// TIA Portal V17 export
// export: Created 2025-03-05T07:58:52.0345726Z, ExportSetting WithDefaults, DisplayName Totally Integrated Automation Portal, DisplayVersion V17 Update 8, DisplayName TIA Portal Openness, DisplayVersion V17 Update 8, DisplayName TIA Portal Version Control Interface, DisplayVersion V17, DisplayName SINAMICS Startdrive Advanced, DisplayVersion V17 SP2, DisplayName SINAMICS Startdrive G110M, G120, G120C, G120D, G120P, G115D, DisplayVersion V17 SP2, DisplayName SINAMICS Startdrive G130, G150, S120, S150, SINAMICS MV, S210, DisplayVersion V17 SP2, DisplayName STEP 7 Professional, DisplayVersion V17 Update 8, DisplayName SINUMERIK ONE STEP 7 Toolbox, DisplayVersion V17 Update 12, DisplayName SINUMERIK 840D sl STEP 7 Toolbox, DisplayVersion V17 Update 12, DisplayName STEP 7 Safety, DisplayVersion V17 Update 6, DisplayName WinCC Advanced, DisplayVersion V17 Update 8
DATA_BLOCK "LBP_HMI"   // DB19
TITLE = Operator panel signals / Señales panel de mando / Bedienfeld-Signale
{ S7_Optimized_Access := 'FALSE'; DB_Accessible_From_OPC_UA := 'FALSE' }
AUTHOR : SINUMERIK
FAMILY : SINUMERIK_ONE
VERSION : 6.15
// Interface between user program and operator panel, contains signals from/to the operating software. / Interfaz entre programa de usuario y panel de mando, contiene señales desde/hacia software operativo. / Schnittstelle zwischen Anwenderprogramm und Bedienfeld, enthält Signale von der/zu der Betriebssoftware.
// stored: AutoNumber false, DBAccessibleFromOPCUA false, DBAccessibleFromWebserver true, InstanceOfName LBP_typeHMI, InstanceOfType UDT, IsOnlyStoredInLoadMemory false, IsWriteProtectedInAS false
"LBP_typeHMI"
   // VAR RETAIN
   //    A_SCLight : Bool;
   //    A_SCDark : Bool;
   //    A_KeyDisable : Bool;
   //    A_ClearCanAl : Bool;
   //    A_ClearRecAl : Bool;
   //    f0_5 : Bool;
   //    A_SafeActionLog : Bool;
   //    A_ActWCS : Bool;
   //    A_PLCExtViewerReject : Bool;
   //    A_PLCExtViewerMode : Bool;
   //    f1_2 : Bool;
   //    f1_3 : Bool;
   //    f1_4 : Bool;
   //    f1_5 : Bool;
   //    f1_6 : Bool;
   //    f1_7 : Bool;
   //    A_1stError1 : Word;
   //    A_1stError2 : Word;
   //    A_ASpi1percent : Byte;
   //    A_ASpi2percent : Byte;
   //    A_MCPChan : Byte;
   //    A_OEM1 : Bool;
   //    A_OEM2 : Bool;
   //    A_AToolMeas : Bool;
   //    f9_3 : Bool;
   //    f9_4 : Bool;
   //    f9_5 : Bool;
   //    f9_6 : Bool;
   //    f9_7 : Bool;
   //    A_Hardkey : Byte;
   //    f11 : Byte;
   //    f12_0 : Bool;
   //    f12_1 : Bool;
   //    A_COM2 : Bool;
   //    A_COM1 : Bool;
   //    A_V24stop : Bool;
   //    A_V24ext : Bool;
   //    A_V24off : Bool;
   //    A_V24on : Bool;
   //    A_TeachDisable : Bool;
   //    f13_1 : Bool;
   //    f13_2 : Bool;
   //    f13_3 : Bool;
   //    f13_4 : Bool;
   //    A_PPdeload : Bool;
   //    A_PPload : Bool;
   //    A_PPsel : Bool;
   //    A_V24Index1 : Byte;
   //    A_V24Index2 : Byte;
   //    A_V24NoFile1 : Byte;
   //    A_V24NoFile2 : Byte;
   //    A_res18 : Byte;
   //    A_res19 : Byte;
   //    f20_0 : Bool;
   //    E_SCDark : Bool;
   //    E_Cancel : Bool;
   //    E_CanCleared : Bool;
   //    E_RecCleared : Bool;
   //    f20_5 : Bool;
   //    E_SimActiv : Bool;
   //    E_ActWCS : Bool;
   //    E_ActivWA : Byte;
   //    E_Chan : Byte;
   //    E_KeybHandl : Bool;
   //    E_DataTransf : Bool;
   //    E_DisplChange : Bool;
   //    f23_3 : Bool;
   //    f23_4 : Bool;
   //    f23_5 : Bool;
   //    f23_6 : Bool;
   //    f23_7 : Bool;
   //    E_ScreenNo : Word;
   //    E_res26_0 : Bool;
   //    E_PPOK : Bool;
   //    E_PPErr : Bool;
   //    E_PPAct : Bool;
   //    f26_4 : Bool;
   //    E_PPdeload : Bool;
   //    E_PPload : Bool;
   //    E_PPsel : Bool;
   //    E_PPError : Byte;
   //    A_PictNo : Int;
   //    A_PictOn : Bool;
   //    A_PictOff : Bool;
   //    f30_2 : Bool;
   //    f30_3 : Bool;
   //    f30_4 : Bool;
   //    f30_5 : Bool;
   //    f30_6 : Bool;
   //    f30_7 : Bool;
   //    E_PictOK : Bool;
   //    E_PictOn : Bool;
   //    E_PictAct : Bool;
   //    E_PictOff : Bool;
   //    E_PictErr : Bool;
   //    f31_5 : Bool;
   //    f31_6 : Bool;
   //    E_NotAct : Bool;
   //    A_FuncNo : Byte;
   //    A_Par1 : Byte;
   //    A_Par2 : Byte;
   //    A_Par3 : Byte;
   //    E_FuncErr : Byte;
   //    f37 : Byte;
   //    f38 : Byte;
   //    f39 : Byte;
   //    res40 : Array[0..9] of Byte;
   //    MMC2 : Struct
   //       A_SCLight : Bool;
   //       A_SCDark : Bool;
   //       A_KeyDisable : Bool;
   //       A_ClearCanAl : Bool;
   //       A_ClearRecAl : Bool;
   //       f0_5 : Bool;
   //       f0_6 : Bool;
   //       A_ActWCS : Bool;
   //       A_PLCExtViewerReject : Bool;
   //       A_PLCExtViewerMode : Bool;
   //       f1_2 : Bool;
   //       f1_3 : Bool;
   //       f1_4 : Bool;
   //       f1_5 : Bool;
   //       f1_6 : Bool;
   //       f1_7 : Bool;
   //       A_1stError1 : Word;
   //       A_1stError2 : Word;
   //       A_ASpi1percent : Byte;
   //       A_ASpi2percent : Byte;
   //       A_MCPChan : Byte;
   //       A_OEM1 : Bool;
   //       A_OEM2 : Bool;
   //       A_AToolMeas : Bool;
   //       f9_3 : Bool;
   //       f9_4 : Bool;
   //       f9_5 : Bool;
   //       f9_6 : Bool;
   //       f9_7 : Bool;
   //       A_Hardkey : Byte;
   //       f11 : Byte;
   //       f12_0 : Bool;
   //       f12_1 : Bool;
   //       A_COM2 : Bool;
   //       A_COM1 : Bool;
   //       A_V24stop : Bool;
   //       A_V24ext : Bool;
   //       A_V24off : Bool;
   //       A_V24on : Bool;
   //       A_TeachDisable : Bool;
   //       f13_1 : Bool;
   //       f13_2 : Bool;
   //       f13_3 : Bool;
   //       f13_4 : Bool;
   //       A_PPdeload : Bool;
   //       A_PPload : Bool;
   //       A_PPsel : Bool;
   //       A_V24Index1 : Byte;
   //       A_V24Index2 : Byte;
   //       A_V24NoFile1 : Byte;
   //       A_V24NoFile2 : Byte;
   //       A_res18 : Byte;
   //       A_res19 : Byte;
   //       f20_0 : Bool;
   //       E_SCDark : Bool;
   //       E_Cancel : Bool;
   //       E_CanCleared : Bool;
   //       E_RecCleared : Bool;
   //       f20_5 : Bool;
   //       E_SimActiv : Bool;
   //       E_ActWCS : Bool;
   //       E_ActivWA : Byte;
   //       E_Chan : Byte;
   //       E_KeybHandl : Bool;
   //       E_DataTransf : Bool;
   //       E_DisplChange : Bool;
   //       f23_3 : Bool;
   //       f23_4 : Bool;
   //       f23_5 : Bool;
   //       f23_6 : Bool;
   //       f23_7 : Bool;
   //       E_ScreenNo : Word;
   //       E_res26_0 : Bool;
   //       E_PPOK : Bool;
   //       E_PPErr : Bool;
   //       E_PPAct : Bool;
   //       f26_4 : Bool;
   //       E_PPdeload : Bool;
   //       E_PPload : Bool;
   //       E_PPsel : Bool;
   //       E_PPError : Byte;
   //       A_PictNo : Int;
   //       A_PictOn : Bool;
   //       A_PictOff : Bool;
   //       f30_2 : Bool;
   //       f30_3 : Bool;
   //       f30_4 : Bool;
   //       f30_5 : Bool;
   //       f30_6 : Bool;
   //       f30_7 : Bool;
   //       E_PictOK : Bool;
   //       E_PictOn : Bool;
   //       E_PictAct : Bool;
   //       E_PictOff : Bool;
   //       E_PictErr : Bool;
   //       f31_5 : Bool;
   //       f31_6 : Bool;
   //       E_NotAct : Bool;
   //       A_FuncNo : Byte;
   //       A_Par1 : Byte;
   //       A_Par2 : Byte;
   //       A_Par3 : Byte;
   //       E_FuncErr : Byte;
   //       f37 : Byte;
   //       f38 : Byte;
   //       f39 : Byte;
   //       res40 : Array[0..9] of Byte;
   //    END_STRUCT;
   //    ONL_REQUEST : Word;
   //    ONL_CONFIRM : Word;
   //    PAR_CLIENT_IDENT : Word;
   //    PAR_MMC_TYP : Byte;
   //    PAR_MSTT_ADR : Byte;
   //    PAR_STATUS : Byte;
   //    PAR_Z_INFO : Byte;
   //    MtoNAlive : Word;
   //    f112 : Byte;
   //    ParOpKeyAdr : Byte;
   //    ParTcuIndex : Byte;
   //    f115 : Byte;
   //    Tcu1KeyAdr : Byte;
   //    Tcu2KeyAdr : Byte;
   //    Tcu1Index : Byte;
   //    Tcu2Index : Byte;
   //    MMC1_CLIENT_IDENT : Word;
   //    MMC1_TYP : Byte;
   //    MMC1_MSTT_ADR : Byte;
   //    MMC1_STATUS : Byte;
   //    MMC1_Z_INFO : Byte;
   //    MMC1_SHIFT_LOCK : Bool;
   //    MMC1_MSTT_SHIFT_LOCK : Bool;
   //    MMC1_ACTIVE_REQ : Bool;
   //    MMC1_ACTIVE_PERM : Bool;
   //    MMC1_ACTIVE_CHANGED : Bool;
   //    MMC1_CHANGED_DENIED : Bool;
   //    MMC1_TCU_SHIFT_LOCK : Bool;
   //    f127 : Byte;
   //    MMC1_TRANS_DB : Word;
   //    MMC2_CLIENT_IDENT : Word;
   //    MMC2_TYP : Byte;
   //    MMC2_MSTT_ADR : Byte;
   //    MMC2_STATUS : Byte;
   //    MMC2_Z_INFO : Byte;
   //    MMC2_SHIFT_LOCK : Bool;
   //    MMC2_MSTT_SHIFT_LOCK : Bool;
   //    MMC2_ACTIVE_REQ : Bool;
   //    MMC2_ACTIVE_PERM : Bool;
   //    MMC2_ACTIVE_CHANGED : Bool;
   //    MMC2_CHANGED_DENIED : Bool;
   //    MMC2_TCU_SHIFT_LOCK : Bool;
   //    f137 : Byte;
   //    MMC2_TRANS_DB : Word;
   //    A_Subtype : Int;
   //    A_Duplo : Int;
   //    A_Ident : String[32];
   //    A_Tnumber : Int;
   //    A_MagazinePlace : Int;
   //    A_MagazinePlaceType : Int;
   //    A_ToolSize_Upper : Byte;
   //    A_ToolSize_Down : Byte;
   //    A_ToolSize_Left : Byte;
   //    A_ToolSize_Right : Byte;
   //    A_Channel : Byte;
   //    A_LoadingPlace : Byte;
   //    A_Magazine : Int;
   //    A_Unit : Byte;
   //    A_NCU_Index : Byte;
   //    A_FileIndex : Int;
   //    A_ActiveEnable : Bool;
   //    A_Override : Bool;
   //    A_LoadTool : Bool;
   //    A_DeleteTool : Bool;
   //    E_Subtype : Int;
   //    E_Duplo : Int;
   //    E_Ident : String[32];
   //    E_Tnumber : Int;
   //    E_ToolState : Int;
   //    E_MagazinePlaceType : Int;
   //    E_ToolSize_Upper : Byte;
   //    E_ToolSize_Down : Byte;
   //    E_ToolSize_Left : Byte;
   //    E_ToolSize_Right : Byte;
   //    E_Magazine : Int;
   //    E_MagazinePlace : Int;
   //    A_ReqMMC1 : Bool;
   //    A_ReqMMC2 : Bool;
   //    A_K_Code : Byte;
   //    E_Done : Bool;
   //    E_Error : Bool;
   //    E_Active : Bool;
   //    f252_3 : Bool;
   //    f252_4 : Bool;
   //    f252_5 : Bool;
   //    f252_6 : Bool;
   //    E_Ident_Ready : Bool;
   //    E_K_CodeError : Byte;
   //    E_Error_Code : Int;
   //    E_Req : Bool;
   //    f257 : Byte;
   //    A_Done : Bool;
   //    A_Error : Bool;
   //    A_Active : Bool;
   //    f258_3 : Bool;
   //    f258_4 : Bool;
   //    f258_5 : Bool;
   //    f258_6 : Bool;
   //    f258_7 : Bool;
   //    E_TDC_Read : Bool;
   //    E_TDC_Write : Bool;
   //    E_TDC_Cancel : Bool;
   //    E_TDC_Read_before_Write : Bool;
   //    f259_4 : Bool;
   //    f259_5 : Bool;
   //    f259_6 : Bool;
   //    f259_7 : Bool;
   //    A_Error_Code : Int;
   //    E_PMagazine : Int;
   //    E_PMagazinePlace : Int;
   //    E_PTnumber : Int;
   //    A_TPMStatus : Int;
   //    A_TPMCounter : Array[1..32] of DInt;
   //    A_HWeelSimOvr : Byte;
   //    f399 : Byte;
   //    A_SimOvr : Int;
   //    A_SimState : Int;
   //    E_HmiUserKey : Array[1..64] of Bool;
   //    A_HmiUserLed : Array[1..64] of Bool;
   //    A_DisableHmiUserKey : Array[1..64] of Bool;
   // END_VAR
BEGIN
END_DATA_BLOCK
